DATA_BLOCK "Sys_DB"
{ S7_Optimized_Access := 'TRUE' }
VERSION : 0.1
NON_RETAIN
"Sys"

BEGIN

END_DATA_BLOCK

